TYPE CamIn_CMD_typ :
STRUCT
	StartSlave : BOOL ;
	DisengageSlave : BOOL ;
END_STRUCT
END_TYPE

(* stored: Version 1.1.0.1, ProductVersion 3.1.4024.3
   DUT CamIn_CMD_typ: Id {f64b2959-9ded-0018-1ee6-bb79d0936808} *)
